(* CODESYS project templatecore.library
   Author: Multiple
   Placeholder: TemplateCore
   Title: TemplateCore
   Version: 2.0.0.2
   Description: Template Framework Code
   Company: TemplateCore Creators

Project tree, tasks and I/O mapping:
  libraries: Tc2_Standard, * (Beckhoff Automation GmbH); Tc2_System, * (Beckhoff Automation GmbH); Tc2_TcpIp, * (Beckhoff Automation GmbH); Tc2_Utilities, * (Beckhoff Automation GmbH); Tc3_Module, * (Beckhoff Automation GmbH)
  DUTs/
    Stats/
      data type Component_Stats
      data type StatsAggregateFIFOBuffer
      data type StatsAggregateRecord
      data type StatsConstants
      data type StatsEvent
      data type StatsEventFIFOBuffer
      data type StatsFailure
      data type StatsFailureFIFOBuffer
      data type StatsFault
      data type StatsFaultFIFOBuffer
      data type StatsShiftAggregateFIFOBuffer
      data type StatsShiftAggregateRecord
    data type Channels
    data type Colors
    data type ComponentIdentifier
    data type Dint100FIFOBuffer
    data type FaultMessage
    data type FrameWork
    data type FrameworkLocal
    data type GeneralMessage
    data type HMIBanner
    data type HMIMessage
    data type HMIMessageBuffer
    data type ID50FIFOBuffer
    data type LREAL100FIFOBuffer
    data type StateTimeStamp
    data type Station
    data type STRING256
    data type TimeStamp
    data type TraceFIFOBuffer
  GVLs/
    global variables GVL
  POUs/
    FrameWork/
      function F_AddMessage [ST]
      function F_FindMessage [ST]
      function block FB_Framework [ST]
      function block FIFO_HMIMessage [ST]: INIT, INSERT, PEEK, REMOVE
    OEE/
      function F_SendEvent [ST]
      function block FIFO_StatsAggregate [ST]: INIT, INSERT, PEEK, PEEKLAST, REMOVE
      function block FIFO_StatsEvent [ST]: INIT, INSERT, PEEK, REMOVE
      function block FIFO_StatsFailureLog [ST]: INIT, INSERT, PEEK, REMOVE
      function block FIFO_StatsFaultLog [ST]: INIT, INSERT, PEEK, REMOVE
      function block FIFO_StatsShiftAggregate [ST]: INIT, INSERT, PEEK, REMOVE
    StateTrace/
      function block FIFO_StateTrace [ST]: INIT, INSERT, PEEK, REMOVE
    TCP Communications/
      function block FB_TCPClient [ST]
    Utility/
      function F_GetTimeStamp [ST]
      function block FB_FileReadSettings [ST]
      function block FB_FileWriteSettings [ST]
      function block FB_Sensor [ST]
      function block FIFO_DINT100 [ST]: INIT, INSERT, PEEK, REMOVE
      function block FIFO_ID50 [ST]: INIT, INSERT, PEEK, REMOVE
      function block FIFO_LREAL100 [ST]: INIT, INSERT, PEEK, REMOVE
      function LEFTBigString [ST]
      function RIGHTBigString [ST]
    program MAIN [ST]
  Version/
    global variables Global_Version
  VISUs/
*)

// DUTs/Stats/Component_Stats
{attribute 'pack_mode' := '1'}
TYPE Component_Stats :
STRUCT
	AggregateInterval : DINT ; (*interval time in minutes*)
	PlannedDowntime : ARRAY [0..2] OF DINT;  (*index corresponds to shift number*)
	StartOfShift : ARRAY [0..2,0..1] OF DINT; (*[shift number],[hour,min]*)
	IdealCycleTime : LREAL; (*cycle time is second*)

	StatsEventFIFO : FIFO_StatsEvent := (Overwrite := TRUE);
	StatsEventBuffer : StatsEventFIFObuffer;
	StatsAggregateFIFO : FIFO_StatsAggregate := (Overwrite := TRUE);
	StatsAggregateBuffer : StatsAggregateFIFOBuffer;
	StatsShiftAggregateFIFO : FIFO_StatsShiftAggregate := (Overwrite := TRUE);
	StatsShiftAggregateBuffer : StatsShiftAggregateFIFOBuffer;
	StatsFaultLog : FIFO_StatsFaultLog := (Overwrite := TRUE);
	StatsFaultLogBuffer : StatsFaultFIFOBuffer;
	StatsFailureLog : FIFO_StatsFailureLog := (Overwrite := TRUE);
	StatsFailureLogBuffer : StatsFailureFIFOBuffer;

	StatsIdealCycleTimeFIFO : FIFO_LREAL100 := (Overwrite := FALSE);
	StatsIdealCycleTimeBuffer : LREAL100FIFOBuffer;
	StatsPartCountFIFO : FIFO_DINT100 := (Overwrite := FALSE);
	StatsPartCountBuffer : Dint100FIFOBuffer;

	Framework : Framework;
END_STRUCT
END_TYPE

// DUTs/Stats/StatsAggregateFIFOBuffer
TYPE StatsAggregateFIFOBuffer :
STRUCT
	Size:DINT := 864; (*3days at 5min*)
	Buffer:ARRAY [0..863] OF StatsAggregateRecord;
END_STRUCT
END_TYPE

// DUTs/Stats/StatsAggregateRecord
TYPE StatsAggregateRecord :
STRUCT
	TimeStamp : TimeStamp;
	OperatorStopTime : LREAL;
	OperatorStopCount : DINT;
	AutoStopTime:LREAL;
	AutoStopCount : DINT;
	WorkTime : LREAL;
	WorkCount: DINT;
	BypassTime: LREAL;
	BypassCount: DINT;
	BlockTime: LREAL;
	BlockCount: DINT;
	StarveTime:LREAL;
	StarveCount:DINT;
	FaultTime:LREAL;
	FaultCount:DINT;
	EmptyTime:LREAL;
	EmptyCount:DINT;
	RetryTime:LREAL;
	RetryCount:DINT;
	MasterTime:LREAL;
	MasterCount:DINT;
	OtherTime:LREAL;
	OtherCount:DINT;
	RejectCount:DINT;
	GoodCount:DINT;
	FirstTimeGoodCount:DINT;
	FirstTimeStartCount:DINT;
	GoodCycleTime:LREAL;
	InitCount:DINT;
	PartsForCurrentCycleTime: DINT;
	Shift : DINT;
END_STRUCT
END_TYPE

// DUTs/Stats/StatsConstants
TYPE StatsConstants :
STRUCT
	Aggregate :DINT := 1;

	OperatorStop : DINT := 100;
	MachineStop : DINT  :=101;
	Working : DINT := 102;
	Bypass : DINT := 103;
	Blocked : DINT := 104;
	Starved : DINT := 105;
	Faulted : DINT :=106;
	FaultAcknowledge : DINT := 107;
	Empty : DINT := 108;
	Retry : DINT := 109;
	Mastering : DINT := 110;

	Failure : DINT := 200;
	Good : DINT := 201;
	FirstTimeGood : DINT := 202;
	FirstTimeStart : DINT := 203;
	Initialize : DINT := 204;

	PartChange : DINT := 300;
	CycleTime : DINT := 301;


END_STRUCT
END_TYPE

// DUTs/Stats/StatsEvent
TYPE StatsEvent :
STRUCT
	TimeStamp : TimeStamp;
	EType : DINT;
	Data : ARRAY[0..4] OF REAL;
	StringData :ARRAY[0..3] OF STRING(80);
END_STRUCT
END_TYPE

// DUTs/Stats/StatsEventFIFOBuffer
{attribute 'pack_mode' := '1'}
TYPE StatsEventFIFOBuffer :
STRUCT
	Size:DINT := 100;
	Buffer:ARRAY[0..99] OF StatsEvent;
END_STRUCT
END_TYPE

// DUTs/Stats/StatsFailure
TYPE StatsFailure :
STRUCT
	TimeStamp : TimeStamp;
	StationID : DINT;
	FailureID : DINT;
	Parameters : STRING;
END_STRUCT
END_TYPE

// DUTs/Stats/StatsFailureFIFOBuffer
TYPE StatsFailureFIFOBuffer :
STRUCT
	Size:UDINT := 500;
	Buffer:ARRAY [0..499] OF StatsFailure;
END_STRUCT
END_TYPE

// DUTs/Stats/StatsFault
TYPE StatsFault:
STRUCT
	TimeStamp : TimeStamp;
	StationID : DINT;
	FaultID : DINT;
	AcknowledgeTime : LREAL;
	Duration : LREAL;
	Data : ARRAY [0..2] OF REAL;
	StringData : ARRAY [0..3] OF STRING;
END_STRUCT
END_TYPE

// DUTs/Stats/StatsFaultFIFOBuffer
TYPE StatsFaultFIFOBuffer :
STRUCT
	Size:UDINT := 500;
	Buffer:ARRAY [0..499] OF StatsFault;
END_STRUCT
END_TYPE

// DUTs/Stats/StatsShiftAggregateFIFOBuffer
TYPE StatsShiftAggregateFIFOBuffer :
STRUCT
	Size:DINT := 270; (*90 days*)
	Buffer:ARRAY [0..269] OF StatsShiftAggregateRecord;
END_STRUCT
END_TYPE

// DUTs/Stats/StatsShiftAggregateRecord
TYPE StatsShiftAggregateRecord :
STRUCT
	AggregateData : StatsAggregateRecord;
	Shift : DINT;
	ShiftStartTimeStamp : TimeStamp;
	AvailableTime : LREAL;
	NetAvailableTime : LREAL;
	TotalDownTime: LREAL;
	PlannedDownTime: LREAL;
	UnplannedDownTime: LREAL;
	OperatingTime : LREAL;
	EquipmentAvailability : LREAL;
	TotalParts: DINT;
	PerformanceEfficiency : LREAL;
	QualityRate : LREAL;
	OverallEquipmentEffectiveness :LREAL;
	CycleTimeAvgSum: LREAL;
	CycleTimeAvgCnt: DINT;
END_STRUCT
END_TYPE

// DUTs/Channels
TYPE Channels :
STRUCT
	Fault :DINT:= 1;
	Attention:DINT := 2;
	General:DINT:= 3;
	FirstFault:DINT:= 4;
END_STRUCT
END_TYPE

// DUTs/Colors
TYPE Colors :
STRUCT
	Red: DINT := 255;
	Green: DINT :=65280;
	Grey: DINT :=8421504;
	Black: DINT := 0;
	Yellow: DINT := 65535;
	Blue: DINT := 16711680;
	White:DINT := 16777215;
END_STRUCT
END_TYPE

// DUTs/ComponentIdentifier
TYPE ComponentIdentifier :
STRUCT
	ID:DINT;
	Name:STRING;
END_STRUCT
END_TYPE

// DUTs/Dint100FIFOBuffer
TYPE Dint100FIFOBuffer :
STRUCT
	Size:DINT := 100;
	Buffer:ARRAY [0..99] OF DINT;
END_STRUCT
END_TYPE

// DUTs/FaultMessage
TYPE FaultMessage :
STRUCT
	Id: DINT;
	Text: STRING256;
	AltText: STRING256;
END_STRUCT
END_TYPE

// DUTs/FrameWork
TYPE FrameWork :
STRUCT
	OnScan:BOOL;
	ResetStart:BOOL;
	ResetDone:BOOL;
	FullInitRequired:BOOL;
	Behavior:DINT;
	ComponentIDRecord: ComponentIdentifier;
END_STRUCT
END_TYPE

// DUTs/FrameworkLocal
TYPE FrameworkLocal :
STRUCT
	AsynchFault: BOOL;
	AsynchFaultReactionComplete: BOOL;
	Attention: BOOL;
	CycleAuto: BOOL;
	CycleFaulted: BOOL;
	CycleManual: BOOL;
	CycleReset: BOOL;
	ManualCycleRequested: BOOL;
	ManualCycleDone: BOOL;
	OKToStop: BOOL;
	SingleStepInhibit: BOOL;
	IgnorSingleStep: BOOL;
	FirstEntry: BOOL;
	LongFaultState: BOOL;
	CycleAutoFallingEdge: F_TRIG;
	CycleResetFallingEdge: F_TRIG;
	CycleManualFallingEdge: F_TRIG;
	State: DINT;
	NextState: DINT;
	LastAutoState: DINT;
	ReEntryState: DINT;
	FaultedState: DINT;
	FaultNumber: DINT;
	LocalFaultID: DINT;
	FullFaultID: DINT;
	tmrState: TON;
	tmrFault: TON;
	StateTimePreset:TIME;
	FaultTimePreset:TIME;
	FaultTimeLong: TIME;
	FaultTimeShort: TIME;
	FaultText: STRING256;
	FaultAltText: STRING256;
	FaultData:StatsFault;
	MsgText: STRING256;
	AltMsgText: STRING256;
	MsgArray: ARRAY [0..99] OF GeneralMessage;
	HMIMsg: HMIMessage;
	StateTimeStamp: StateTimeStamp;
	CurrentTime: TimeStamp;
	Name:STRING(30);
	AltName:STRING(30);
	pStateTraceBuffer: POINTER TO TraceFIFOBuffer;
	pStateTraceFifo: POINTER TO FIFO_StateTrace;
	pStats: POINTER TO Component_Stats;
END_STRUCT
END_TYPE

// DUTs/GeneralMessage
TYPE GeneralMessage :
STRUCT
	Id: DINT;
	BitNumber: DINT;
	Text: STRING;
	AltText:STRING;
END_STRUCT
END_TYPE

// DUTs/HMIBanner
TYPE HMIBanner :
STRUCT
	Text:STRING256;
	AltText:STRING256;
	Color:DINT;
END_STRUCT
END_TYPE

// DUTs/HMIMessage
TYPE HMIMessage :
STRUCT
	Channel: DINT;
	Color: DINT;
	Text: STRING256;
	AltText: STRING256;
END_STRUCT
END_TYPE

// DUTs/HMIMessageBuffer
TYPE HMIMessageBuffer :
STRUCT
	Size:DINT := 100;
	Buffer:ARRAY [0..99] OF HMIMessage;
END_STRUCT
END_TYPE

// DUTs/ID50FIFOBuffer
TYPE ID50FIFOBuffer :
STRUCT
	Size:DINT := 50;
	Buffer:ARRAY [0..49] OF ComponentIdentifier;
END_STRUCT
END_TYPE

// DUTs/LREAL100FIFOBuffer
TYPE LREAL100FIFOBuffer :
STRUCT
	Size:DINT := 100;
	Buffer:ARRAY [0..99] OF LREAL;
END_STRUCT
END_TYPE

// DUTs/StateTimeStamp
TYPE StateTimeStamp :
STRUCT
	Station:DINT;
	ID:DINT;
	State:DINT;
	TimeLo:UDINT;
	TimeHi:UDINT;
END_STRUCT
END_TYPE

// DUTs/Station
TYPE Station :
STRUCT
	CycleAuto:BOOL;
	CycleReset:BOOL;
	CycleManual:BOOL;
	CycleStopped:BOOL;
	CycleFaulted:BOOL;
	OKToStop:BOOL;
	OKForManual:BOOL;
	StopRequest:BOOL;
	EmergencyStop:BOOL;
	UnlatchFaults:BOOL;
	FaultReset:BOOL;
	FullInitRequired:BOOL;
	ResetDone:BOOL;
	SingleStep:BOOL;
	StepAdvance:BOOL;
	DryCycle:BOOL;
	Attention:BOOL;
	MachineStopRqst:BOOL;

	hiCycleStart:BOOL;
	hiCycleStop:BOOL;
	hiFaultAck:BOOL;
	hiFaultReset:BOOL;
	hiStationReset:BOOL;
	hiSingleStepOn:BOOL;
	hiSingleStepOff:BOOL;
	hiSingleStepAdvance:BOOL;
	hiManualMode:BOOL;
	hiLampTest:BOOL;
	hoStationResetRequired:BOOL;

	StationID:DINT;
	MachineID:DINT;
	FirstFault:StatsFault;
	PreviousStationID:DINT;
	NextStationID:DINT;
	HMIMessageFIFO: FIFO_HMIMessage;
	HMIMessageBuffer: HMIMessageBuffer;
	StationMessage:HMIBanner;
	OperatorMessage:HMIBanner;
	b500msPulse: BOOL;

	FaultedFIFO: FIFO_ID50;
	FaultedFIFOBuffer: ID50FIFOBuffer;
	NotOKtoStopFIFO: FIFO_ID50;
	NotOKToStopFIFOBuffer:ID50FIFOBuffer;
	AttentionRequiredFIFO: FIFO_ID50;
	AttentionRequiredFIFOBuffer: ID50FIFOBuffer;
	CycleManualFIFO: FIFO_ID50;
	CycleManualFIFOBuffer:ID50FIFOBuffer;

END_STRUCT
END_TYPE

// DUTs/STRING256
TYPE STRING256 :STRING[256];

END_TYPE

// DUTs/TimeStamp
TYPE TimeStamp :
STRUCT
	CurrentValue : T_ULarge_Integer;
	DateTime: TIMESTRUCT;
END_STRUCT
END_TYPE

// DUTs/TraceFIFOBuffer
TYPE TraceFIFOBuffer :
STRUCT
	Size:DINT := 1000;
	Buffer:ARRAY [0..999] OF StateTimeStamp;
END_STRUCT
END_TYPE

// GVLs/GVL
{attribute 'qualified_only'}
VAR_GLOBAL
	cColor:Colors;
	cChannel:Channels;
	cNullString:STRING;
	cEmptyHMIMessage: HMIMessage;(* ~(OPC:1:available for OPC-clients) *)
	gTimeZoneOffsetFromUTC: DINT := 0;
	gFirstScan:BOOL;
	gCurrentTime : TimeStamp;
END_VAR

// Version/Global_Version
{attribute 'TcGenerated'}
// This function has been automatically generated from the project information.
VAR_GLOBAL CONSTANT
	{attribute 'const_non_replaced'}
	{attribute 'linkalways'}
	stLibVersion_TemplateCore : ST_LibVersion := (iMajor := 2, iMinor := 0, iBuild := 0, iRevision := 2, sVersion := '2.0.0.2');
END_VAR

// POUs/FrameWork/F_AddMessage
FUNCTION F_AddMessage : BOOL
VAR_INPUT
	pStation:  POINTER TO Station;
	Text:STRING256	;
	AltText:STRING256;
	Color:DINT;
	Channel:DINT;
END_VAR
VAR
	StationAddress:DINT;
	HMIMsg:HMIMessage;

END_VAR

HMIMsg.Text := Text;
HMIMsg.AltText := AltText;
HMIMsg.Color := Color;
HMIMsg.Channel := Channel;
pStation^.HMIMessageFIFO.INSERT(pFIFO:=ADR(pStation^.HMIMessageBuffer), in :=HMIMsg);

END_FUNCTION

// POUs/FrameWork/F_FindMessage
FUNCTION F_FindMessage : GeneralMessage
VAR_INPUT
	pLocal: POINTER TO FrameworkLocal;
	State:DINT;
	ID: DINT;
END_VAR
VAR
	Msg:GeneralMessage;
	idx:DINT;
	length:DINT;
END_VAR

length := SIZEOF(pLocal^.MsgArray) / SIZEOF(Msg);
Msg.Text  :='**No message text**';
Msg.AltText :='**No alt message text**';
FOR idx :=0 TO (length-1) DO
	IF pLocal^.MsgArray[idx].Id = (State * 10 + ID) THEN
		Msg := pLocal^.MsgArray[idx];
		EXIT;
	END_IF
END_FOR
F_FindMessage := Msg;

END_FUNCTION

// POUs/FrameWork/FB_Framework
FUNCTION_BLOCK FB_Framework
VAR_INPUT
	pFrameWork: POINTER TO FrameWork;
	pLocal: POINTER TO FrameworkLocal;
	pStation: POINTER TO Station;
END_VAR

VAR_OUTPUT
END_VAR

VAR
	InitialScan: R_TRIG;
	ActiveStationID: DINT;
	Msg:GeneralMessage;
	cChannel: Channels;
END_VAR

VAR_STAT CONSTANT
	cColor: Colors;
END_VAR

(****************************************************************************
* Framework Post-Sequence Logic, DO NOT modify this section *
*****************************************************************************)

InitialScan(CLK := TRUE);
IF InitialScan.Q THEN
        pLocal^.State := 9999;
        pLocal^.NextState := 5000;
END_IF

(*  Fault Logic  *)
pLocal^.tmrFault(IN := (NOT pLocal^.OKToStop AND NOT pLocal^.FirstEntry AND NOT pLocal^.SingleStepInhibit  AND
				(pLocal^.CycleAuto OR pLocal^.CycleReset OR pLocal^.CycleManual)), PT := pLocal^.FaultTimePreset);
IF pLocal^.FaultNumber  > 0 THEN
	IF  NOT pLocal^.CycleFaulted THEN
		pLocal^.CycleFaulted := TRUE;
		pLocal^.FaultedState := pLocal^.state;
		IF (NOT pLocal^.AsynchFault) OR pLocal^.AsynchFaultReactionComplete THEN
			Msg := F_FindMessage(pLocal,  pLocal^.State, pLocal^.FaultNumber);
			pLocal^.FaultData.FaultID := pFrameWork^.ComponentIDRecord.ID * 100000 + pLocal^.state*10 + pLocal^.FaultNumber;
		ELSE
			Msg := F_FindMessage(pLocal,  0, pLocal^.FaultNumber);
			pLocal^.FaultData.FaultID := pFrameWork^.ComponentIDRecord.ID * 100000 + pLocal^.FaultNumber;
		END_IF
		pLocal^.MsgText :=  'Fault: ';
		pLocal^.AltMsgText  := 'AltFault: ';
		pLocal^.MsgText := CONCAT(pLocal^.MsgText,DINT_TO_STRING(pLocal^.FaultData.FaultID));
		pLocal^.MsgText := CONCAT(pLocal^.MsgText,' ');
		pLocal^.MsgText := CONCAT(pLocal^.MsgText, pLocal^.Name);
		pLocal^.MsgText := CONCAT(pLocal^.MsgText,' -  ');
		pLocal^.MsgText := CONCAT(pLocal^.MsgText, Msg.Text);
		pLocal^.AltMsgText := CONCAT(pLocal^.AltMsgText,DINT_TO_STRING(pLocal^.FaultData.FaultID));
		pLocal^.AltMsgText := CONCAT(pLocal^.AltMsgText,' ');
		pLocal^.AltMsgText := CONCAT(pLocal^.AltMsgText, pLocal^.AltName);
		pLocal^.AltMsgText := CONCAT(pLocal^.MsgText,' -  ');
		pLocal^.AltMsgText:=CONCAT(pLocal^.AltMsgText, Msg.AltText);
		F_AddMessage(pStation, pLocal^.MsgText, pLocal^.AltMsgText, cColor.Red, cChannel.Fault);
		IF pStation^.FirstFault.FaultID = 0 THEN
			pStation^.FirstFault := pLocal^.FaultData;
			pStation^.FirstFault.StationID  := pStation^.StationID;
			pStation^.FirstFault.StringData[0] :=pLocal^.MsgText;
			pStation^.FirstFault.StringData[1] :=pLocal^.AltMsgText;
		END_IF
	END_IF
END_IF

(*END fault logic*)

(***************************************************************************
* Framework Pre-Sequence Logic, DO NOT modify this section *
****************************************************************************)

IF pLocal^.NextState <> pLocal^.state THEN
	pLocal^.FirstEntry := TRUE;
	pLocal^.state := pLocal^.NextState;
	pLocal^.tmrState(IN:=FALSE); (*clear timer if state changes*)

	pLocal^.CurrentTime := GVL.gCurrentTime;
	pLocal^.StateTimeStamp.ID := pFrameWork^.ComponentIDRecord.ID;
	pLocal^.StateTimeStamp.State := pLocal^.State;
	pLocal^.StateTimeStamp.TimeHi := pLocal^.CurrentTime.CurrentValue.dwHighPart;
	pLocal^.StateTimeStamp.TimeLo:= pLocal^.CurrentTime.CurrentValue.dwLowPart;
	pLocal^.pStateTraceFifo^.INSERT(pFIFO := pLocal^.pStateTraceBuffer, in := pLocal^.StateTimeStamp);
ELSE
	pLocal^.FirstEntry := FALSE;
	pLocal^.tmrState(IN:=TRUE,PT:=pLocal^.StateTimePreset);
END_IF

(*On the falling edge of CycleAuto, grab the current state as LastAutoState.
    Also, set the default ReEntryState to the LastAutoState so that we pick back up where 
    we left off after a simple cycle stop / cycle start.
    Set State to 5000, the Idle state. *)

pLocal^.CycleAutoFallingEdge(CLK:=pLocal^.CycleAuto);
IF pLocal^.CycleAutoFallingEdge.Q THEN
	pLocal^.LastAutoState := pLocal^.State;
	pLocal^.ReEntryState := pLocal^.LastAutoState;
	pLocal^.NextState := 5000;
END_IF

(* On the falling edge of CycleReset, set State to 5000, the Idle state.   *)
pLocal^.CycleResetFallingEdge(Clk:=pLocal^.CycleReset);
IF pLocal^.CycleResetFallingEdge.Q THEN
	pLocal^.NextState := 5000;
END_IF

(* On the falling edge of CycleManual, set State to 5000, the Idle state.  *)
pLocal^.CycleManualFallingEdge(Clk:=pLocal^.CycleManual);
IF pLocal^.CycleManualFallingEdge.Q THEN
	pLocal^.NextState := 5000;
END_IF

pLocal^.CycleAuto:=pStation^.CycleAuto AND NOT pLocal^.CycleFaulted;
pLocal^.CycleReset := pStation^.CycleReset AND NOT pLocal^.CycleFaulted;
pLocal^.CycleManual := pLocal^.ManualCycleRequested AND (NOT pLocal^.ManualCycleDone) AND (NOT pStation^.CycleFaulted);
pLocal^.SingleStepInhibit := pStation^.SingleStep AND NOT pStation^.StepAdvance AND NOT pLocal^.IgnorSingleStep;

IF pStation^.UnlatchFaults THEN
	pLocal^.CycleFaulted := FALSE;
	pLocal^.FaultNumber := 0;
END_IF

IF pLocal^.CycleFaulted THEN
	pStation^.FaultedFIFO.INSERT(pFIFO := ADR(pStation^.FaultedFIFOBuffer), in:=pFrameWork^.ComponentIDRecord);
END_IF
IF pLocal^.CycleManual THEN
	pStation^.CycleManualFIFO.INSERT(pFIFO := ADR(pStation^.CycleManualFIFOBuffer), in:=pFrameWork^.ComponentIDRecord);
END_IF
IF pLocal^.Attention THEN
	pStation^.AttentionRequiredFIFO.INSERT(pFIFO := ADR(pStation^.AttentionRequiredFIFOBuffer), in:=pFrameWork^.ComponentIDRecord);
END_IF
IF NOT pLocal^.OKToStop THEN
	pStation^.NotOKtoStopFIFO.INSERT(pFIFO := ADR(pStation^.NotOKtoStopFIFOBuffer), in:=pFrameWork^.ComponentIDRecord);
END_IF
pLocal^.OKToStop := FALSE;
(*END of framework*)

END_FUNCTION_BLOCK

// POUs/FrameWork/FIFO_HMIMessage
FUNCTION_BLOCK FIFO_HMIMessage
VAR_INPUT
	Overwrite	: BOOL;
	pFIFO		: POINTER TO HMIMessageBuffer;
	in			: HMIMessage;
END_VAR
VAR_OUTPUT
	Err		: BOOL;
	Count	: DINT;
	Full		: BOOL;
	out		: HMIMessage;
END_VAR
VAR
	Head : DINT;
	Tail: DINT;
	Idx: DINT;
END_VAR

;

ACTION INIT:
idx := pFIFO^.Size * SIZEOF(in);
MEMSET(ADR( pFIFO^.Buffer[0]), 0, DINT_TO_UDINT(idx));
MEMSET(ADR(in),0,SIZEOF(in));
MEMSET(ADR(out),0,SIZEOF(out));
Count:=0;
Head:=0;
Tail:=0;
Full:=0;
Err:=0;
END_ACTION

ACTION INSERT:
Err := 0;
IF (Full AND Overwrite) OR NOT Full THEN
	pFIFO^.buffer[Head]:=in;
	Head := Head + 1;
	IF Head = pFIFO^.Size THEN
		Head:=0;
	END_IF
	IF Full THEN
		Tail := Tail +1;
		IF Tail = pFIFO^.Size THEN
			Tail :=0;
		END_IF
	ELSE
		Count := Count  +1;
	END_IF
ELSE
	err:=1;
END_IF
Full := (Head = Tail);
END_ACTION

ACTION PEEK:
err:=0;
IF Full OR (Tail <> Head) THEN
	out := pFIFO^.buffer[Tail];
ELSE
	err:=1; (*fifo is empty*)
END_IF
END_ACTION

ACTION REMOVE:
err:=0;
IF NOT Full AND (Head = Tail) THEN
	(*empty*)
	err:=1;
ELSE
	out := pFIFO^.Buffer[Tail];
	MEMSET(ADR(pFIFO^.buffer[Tail]), 0, SIZEOF (in));
	Tail := Tail +1;
	Count := Count  - 1;
	IF Tail = pFIFO^.Size THEN
		Tail := 0;
	END_IF
	Full := 0;
END_IF
END_ACTION

END_FUNCTION_BLOCK

// POUs/OEE/F_SendEvent
FUNCTION F_SendEvent : BOOL
VAR_INPUT
	pStatsFIFO	: POINTER TO FIFO_StatsEvent;
	pBuffer		: POINTER TO StatsEventFIFOBuffer;
	pEvent		: POINTER TO StatsEvent;
END_VAR
VAR
	CurrentTime: TimeStamp;
END_VAR

pEvent^.TimeStamp:= GVL.gCurrentTime;
pStatsFIFO^.INSERT(pFIFO:=pBuffer, in:= pEvent^);
MEMSET(pEvent,0,SIZEOF(pEvent^));

END_FUNCTION

// POUs/OEE/FIFO_StatsEvent
{attribute 'pack_mode' := '1'}
FUNCTION_BLOCK FIFO_StatsEvent
VAR_INPUT
	Overwrite	: BOOL;
	pFIFO		: POINTER TO StatsEventFIFOBuffer;
	in			: StatsEvent;
END_VAR
VAR_OUTPUT
	Err		: BOOL;
	Count	: DINT;
	Full		: BOOL;
	out		: StatsEvent;
END_VAR
VAR
	Head : DINT;
	Tail: DINT;
	Idx: DINT;
END_VAR

ACTION INIT:
Idx := pFIFO^.Size * SIZEOF(in);
MEMSET(ADR( pFIFO^.Buffer[0]), 0, DINT_TO_UDINT(idx));
MEMSET(ADR(in),0,SIZEOF(in));
MEMSET(ADR(out),0,SIZEOF(out));
Count:=0;
Head:=0;
Tail:=0;
Full:=0;
Err:=0;
END_ACTION

ACTION INSERT:
Err := 0;
IF (Full AND Overwrite) OR NOT Full THEN
	pFIFO^.buffer[Head]:=in;
	Head := Head + 1;
	IF Head = pFIFO^.Size THEN
		Head:=0;
	END_IF
	IF Full THEN
		Tail := Tail +1;
		IF Tail = pFIFO^.Size THEN
			Tail :=0;
		END_IF
	ELSE
		Count := Count  +1;
	END_IF
ELSE
	err:=1;
END_IF
Full := (Head = Tail);
END_ACTION

ACTION PEEK:
err:=0;
IF Full OR (Tail <> Head) THEN
	out := pFIFO^.buffer[Tail];
ELSE
	err:=1; (*fifo is empty*)
END_IF
END_ACTION

ACTION REMOVE:
err:=0;
IF NOT Full AND (Head = Tail) THEN
	(*empty*)
	err:=1;
ELSE
	out := pFIFO^.Buffer[Tail];
	MEMSET(ADR(pFIFO^.buffer[Tail]), 0, SIZEOF (in));
	Tail := Tail +1;
	Count := Count  - 1;
	IF Tail = pFIFO^.Size THEN
		Tail := 0;
	END_IF
	Full := 0;
END_IF
END_ACTION

END_FUNCTION_BLOCK

// POUs/OEE/FIFO_StatsAggregate
{attribute 'pack_mode' := '1'}
FUNCTION_BLOCK FIFO_StatsAggregate
VAR_INPUT
	Overwrite	: BOOL;
	pFIFO		: POINTER TO StatsAggregateFIFOBuffer;
	in			: StatsAggregateRecord;
END_VAR
VAR_OUTPUT
	Err		: BOOL;
	Count	: DINT;
	Full		: BOOL;
	out		: StatsAggregateRecord;
END_VAR
VAR
	Head : DINT;
	Tail: DINT;
	Idx: DINT;
END_VAR

ACTION INIT:
idx := pFIFO^.Size * SIZEOF(in);
MEMSET(ADR( pFIFO^.Buffer[0]), 0, DINT_TO_UDINT(idx));
MEMSET(ADR(in),0,SIZEOF(in));
MEMSET(ADR(out),0,SIZEOF(out));
Count:=0;
Head:=0;
Tail:=0;
Full:=0;
Err:=0;
END_ACTION

ACTION INSERT:
Err := 0;
IF (Full AND Overwrite) OR NOT Full THEN
	pFIFO^.buffer[Head]:=in;
	Head := Head + 1;
	IF Head = pFIFO^.Size THEN
		Head:=0;
	END_IF
	IF Full THEN
		Tail := Tail +1;
		IF Tail = pFIFO^.Size THEN
			Tail :=0;
		END_IF
	ELSE
		Count := Count  +1;
	END_IF
ELSE
	err:=1;
END_IF
Full := (Head = Tail);
END_ACTION

ACTION PEEK:
err:=0;
IF Full OR (Tail <> Head) THEN
	out := pFIFO^.buffer[Head];
ELSE
	err:=1; (*fifo is empty*)
END_IF
END_ACTION

ACTION PEEKLAST:
err:=0;
IF Full OR (Tail <> Head) THEN
	out := pFIFO^.buffer[Tail];
ELSE
	err:=1; (*fifo is empty*)
END_IF
END_ACTION

ACTION REMOVE:
err:=0;
IF NOT Full AND (Head = Tail) THEN
	(*empty*)
	err:=1;
ELSE
	out := pFIFO^.Buffer[Tail];
	MEMSET(ADR(pFIFO^.buffer[Tail]), 0, SIZEOF (in));
	Tail := Tail +1;
	Count := Count  - 1;
	IF Tail = pFIFO^.Size THEN
		Tail := 0;
	END_IF
	Full := 0;
END_IF
END_ACTION

END_FUNCTION_BLOCK

// POUs/OEE/FIFO_StatsFailureLog
FUNCTION_BLOCK FIFO_StatsFailureLog
VAR_INPUT
	Overwrite	: BOOL;
	pFIFO		: POINTER TO StatsFailureFIFOBuffer;
	in			: StatsFailure;
END_VAR
VAR_OUTPUT
	Err		: BOOL;
	Count	: DINT;
	Full		: BOOL;
	out		: StatsFailure;
END_VAR
VAR
	Head : DINT;
	Tail: DINT;
	Idx: DINT;
END_VAR

ACTION INIT:
idx := UDINT_TO_DINT(pFIFO^.Size * SIZEOF(in));
MEMSET(ADR( pFIFO^.Buffer[0]), 0, DINT_TO_UDINT(idx));
MEMSET(ADR(in),0,SIZEOF(in));
MEMSET(ADR(out),0,SIZEOF(out));
Count:=0;
Head:=0;
Tail:=0;
Full:=0;
Err:=0;
END_ACTION

ACTION INSERT:
Err := 0;
IF (Full AND Overwrite) OR NOT Full THEN
	pFIFO^.buffer[Head]:=in;
	Head := Head + 1;
	IF Head = UDINT_TO_DINT(pFIFO^.Size) THEN
		Head:=0;
	END_IF
	IF Full THEN
		Tail := Tail +1;
		IF Tail = UDINT_TO_DINT(pFIFO^.Size) THEN
			Tail :=0;
		END_IF
	ELSE
		Count := Count  +1;
	END_IF
ELSE
	err:=1;
END_IF
Full := (Head = Tail);
END_ACTION

ACTION PEEK:
err:=0;
IF Full OR (Tail <> Head) THEN
	out := pFIFO^.buffer[Tail];
ELSE
	err:=1; (*fifo is empty*)
END_IF
END_ACTION

ACTION REMOVE:
err:=0;
IF NOT Full AND (Head = Tail) THEN
	(*empty*)
	err:=1;
ELSE
	out := pFIFO^.Buffer[Tail];
	MEMSET(ADR(pFIFO^.buffer[Tail]), 0, SIZEOF (in));
	Tail := Tail +1;
	Count := Count  - 1;
	IF Tail = UDINT_TO_DINT(pFIFO^.Size) THEN
		Tail := 0;
	END_IF
	Full := 0;
END_IF
END_ACTION

END_FUNCTION_BLOCK

// POUs/OEE/FIFO_StatsFaultLog
FUNCTION_BLOCK FIFO_StatsFaultLog
VAR_INPUT
	Overwrite	: BOOL;
	pFIFO		: POINTER TO StatsFaultFIFOBuffer;
	in			: StatsFault;
END_VAR
VAR_OUTPUT
	Err		: BOOL;
	Count	: DINT;
	Full		: BOOL;
	out		: StatsFault;
END_VAR
VAR
	Head : DINT;
	Tail: DINT;
	Idx: DINT;
END_VAR

ACTION INIT:
idx := UDINT_TO_DINT(pFIFO^.Size * SIZEOF(in));
MEMSET(ADR( pFIFO^.Buffer[0]), 0, DINT_TO_UDINT(idx));
MEMSET(ADR(in),0,SIZEOF(in));
MEMSET(ADR(out),0,SIZEOF(out));
Count:=0;
Head:=0;
Tail:=0;
Full:=0;
Err:=0;
END_ACTION

ACTION INSERT:
Err := 0;
IF (Full AND Overwrite) OR NOT Full THEN
	pFIFO^.buffer[Head]:=in;
	Head := Head + 1;
	IF Head = UDINT_TO_DINT(pFIFO^.Size) THEN
		Head:=0;
	END_IF
	IF Full THEN
		Tail := Tail +1;
		IF Tail = UDINT_TO_DINT(pFIFO^.Size) THEN
			Tail :=0;
		END_IF
	ELSE
		Count := Count  +1;
	END_IF
ELSE
	err:=1;
END_IF
Full := (Head = Tail);
END_ACTION

ACTION PEEK:
err:=0;
IF Full OR (Tail <> Head) THEN
	out := pFIFO^.buffer[Tail];
ELSE
	err:=1; (*fifo is empty*)
END_IF
END_ACTION

ACTION REMOVE:
err:=0;
IF NOT Full AND (Head = Tail) THEN
	(*empty*)
	err:=1;
ELSE
	out := pFIFO^.Buffer[Tail];
	MEMSET(ADR(pFIFO^.buffer[Tail]), 0, SIZEOF (in));
	Tail := Tail +1;
	Count := Count  - 1;
	IF Tail = UDINT_TO_DINT(pFIFO^.Size) THEN
		Tail := 0;
	END_IF
	Full := 0;
END_IF
END_ACTION

END_FUNCTION_BLOCK

// POUs/OEE/FIFO_StatsShiftAggregate
FUNCTION_BLOCK FIFO_StatsShiftAggregate
VAR_INPUT
	Overwrite	: BOOL;
	pFIFO		: POINTER TO StatsShiftAggregateFIFOBuffer;
	in			: StatsShiftAggregateRecord;
	PeekCnt		: DINT;
END_VAR
VAR_OUTPUT
	Err		: BOOL;
	Count	: DINT;
	Full		: BOOL;
	out		: StatsShiftAggregateRecord;
END_VAR
VAR
	Head : DINT;
	Tail: DINT;
	Idx: DINT;

	PeekHead: DINT;
	PeekTail: DINT;
END_VAR

ACTION INIT:
idx := pFIFO^.Size * SIZEOF(in);
MEMSET(ADR( pFIFO^.Buffer[0]), 0, DINT_TO_UDINT(idx));
MEMSET(ADR(in),0,SIZEOF(in));
MEMSET(ADR(out),0,SIZEOF(out));
Count:=0;
Head:=0;
Tail:=0;
Full:=0;
Err:=0;
END_ACTION

ACTION INSERT:
idx := (pFIFO^.Size) * SIZEOF(in);
MEMSET(ADR( pFIFO^.Buffer[0]), 0, DINT_TO_UDINT(idx));
MEMSET(ADR(in),0,SIZEOF(in));
MEMSET(ADR(out),0,SIZEOF(out));
Count:=0;
Head:=0;
Tail:=0;
Full:=0;
Err:=0;
END_ACTION

ACTION PEEK:
err:=0;

PeekHead := Head;
PeekTail := Tail;
FOR Idx := 0 TO PeekCnt DO

	IF NOT Full AND (PeekHead = PeekTail) THEN
		(*empty*)
		err:=1;
	ELSE
		out := pFIFO^.Buffer[PeekTail];
		PeekTail := PeekTail +1;

		IF PeekTail = pFIFO^.Size THEN
			PeekTail := 0;
		END_IF
		Full := 0;
	END_IF
END_FOR

PeekCnt := 0;
END_ACTION

ACTION REMOVE:
err:=0;
IF NOT Full AND (Head = Tail) THEN
	(*empty*)
	err:=1;
ELSE
	out := pFIFO^.Buffer[Tail];
	MEMSET(ADR(pFIFO^.buffer[Tail]), 0, SIZEOF (in));
	Tail := Tail +1;
	Count := Count  - 1;
	IF Tail = pFIFO^.Size THEN
		Tail := 0;
	END_IF
	Full := 0;
END_IF
END_ACTION

END_FUNCTION_BLOCK

// POUs/StateTrace/FIFO_StateTrace
FUNCTION_BLOCK FIFO_StateTrace
VAR_INPUT
	Overwrite	: BOOL;
	pFIFO		: POINTER TO TraceFIFOBuffer;
	in			: StateTimeStamp;
END_VAR
VAR_OUTPUT
	Err		: BOOL;
	Count	: DINT;
	Full		: BOOL;
	out		: StateTimeStamp;
END_VAR
VAR
	Head : DINT;
	Tail: DINT;
	Idx: DINT;
END_VAR

ACTION INIT:
idx := pFIFO^.Size * SIZEOF(in);
MEMSET(ADR( pFIFO^.Buffer[0]), 0, DINT_TO_UDINT(idx));
MEMSET(ADR(in),0,SIZEOF(in));
MEMSET(ADR(out),0,SIZEOF(out));
Count:=0;
Head:=0;
Tail:=0;
Full:=0;
Err:=0;
END_ACTION

ACTION INSERT:
Err := 0;
IF (Full AND Overwrite) OR NOT Full THEN
	pFIFO^.buffer[Head]:=in;
	Head := Head + 1;
	IF Head = pFIFO^.Size THEN
		Head:=0;
	END_IF
	IF Full THEN
		Tail := Tail +1;
		IF Tail = pFIFO^.Size THEN
			Tail :=0;
		END_IF
	ELSE
		Count := Count  +1;
	END_IF
ELSE
	err:=1;
END_IF
Full := (Head = Tail);
END_ACTION

ACTION PEEK:
err:=0;
IF Full OR (Tail <> Head) THEN
	out := pFIFO^.buffer[Tail];
ELSE
	err:=1; (*fifo is empty*)
END_IF
END_ACTION

ACTION REMOVE:
err:=0;
IF NOT Full AND (Head = Tail) THEN
	(*empty*)
	err:=1;
ELSE
	out := pFIFO^.Buffer[Tail];
	MEMSET(ADR(pFIFO^.buffer[Tail]), 0, SIZEOF (in));
	Tail := Tail +1;
	Count := Count  - 1;
	IF Tail = pFIFO^.Size THEN
		Tail := 0;
	END_IF
	Full := 0;
END_IF
END_ACTION

END_FUNCTION_BLOCK

// POUs/TCP Communications/FB_TCPClient
FUNCTION_BLOCK FB_TCPClient
VAR_INPUT
	sRemoteHost: STRING(15);
	nRemotePort:UDINT;
	bConnect:BOOL;
	bSend:BOOL;
	bReceived:BOOL;
	bClearError: BOOL;
	bFlush : BOOL;
	pReceiveBuffer : POINTER TO ARRAY[0..4095] OF USINT;
	pTransmitBuffer : POINTER TO ARRAY[0..4095] OF USINT;
	TransmitLength : DINT;
	pMessageEOF : POINTER TO ARRAY [0..11] OF USINT;
	EOFLength : DINT;
	MessageLength : DINT;
END_VAR
VAR_OUTPUT
	bConnected:BOOL;
	bTransmitComplete:BOOL;
	bError:BOOL;
	bDataAvailable:BOOL;
	nErrorID:DINT;
	sErrorText:STRING(80);
	nReceiveLength:DINT;
	bFlushComplete : BOOL;
END_VAR
VAR
	(*Standard Framework Tags*)
	State: DINT;
	LastState: DINT;
	FaultNumber: DINT;
	FaultedState: DINT;
	FirstEntry: BOOL;
	tmrState: TON;
	MsgText: STRING256;
	AltMsgText:STRING256;
	(*End of Standard Framework Tags*)

	MsgIn: ARRAY[0..4095] OF USINT; (*STRING(4096);*)
	InBuffer: ARRAY[0..12287] OF USINT; (*STRING(12288);*)
	TempBuffer:ARRAY[0..12287] OF USINT;
	InBufferDataLength:DINT :=0;
	pInBuffer:POINTER TO STRING(12288); (*used only to view data easier for debug*)
  	tState120Timer:TON;
	tState200Timer:TON;
	tState500Timer:TON;
	Mode : DINT;
	index : DINT;
	EOFIndex : DINT;
	FindState : DINT;

	hSocketHandle:T_HSOCKET;
	fbSocketConnect : FB_SocketConnect;
	fbSocketClose : FB_SocketClose;
	fbSocketCloseAll : FB_SocketCloseAll;
	fbSocketReceive :FB_SocketReceive;
	fbSocketSend :FB_SocketSend;

END_VAR

VAR CONSTANT
	cEOF : DINT := 1;
	cFixedLength :DINT := 2;
	cContinuous : DINT := 3;
END_VAR

(*If State Change, capture rising edge with FirstEntry.*)
IF State <> LastState THEN
	FirstEntry := TRUE;
	tmrState(IN:=FALSE); (*clear timer if state changes*)
	LastState := State;
ELSIF FirstEntry THEN
	FirstEntry := FALSE;
END_IF

IF EOFLength > 0 THEN
	Mode := cEOF;
ELSIF MessageLength > 0 THEN
	Mode := cFixedLength;
ELSE
	Mode := cContinuous;
END_IF


(**********************
* Sequence logic  *
***********************)
CASE State OF

0:	(*Idle*)
	IF FirstEntry THEN
		bConnected := FALSE;
		bDataAvailable := FALSE;
		bFlushComplete := FALSE;
	END_IF
	IF bConnect AND NOT bError THEN
		State := 100;
	ELSIF bClearError THEN
		bError := FALSE;
		nErrorID := 0;
		sErrorText := GVL.cNullString;
	END_IF

100:	(*Check Parameters*)
	IF sRemoteHost = GVL.cNullString OR nRemotePort = 0 THEN
		bError := TRUE;
		sErrorText:='Invalid connect parameters';
	END_IF
	IF NOT bError THEN
		State := 110;
	ELSE
		State := 0;
	END_IF

110:	(*Connect*)
	IF FirstEntry THEN
		fbSocketConnect(bExecute := FALSE);
		fbSocketConnect(
			sSrvNetId := GVL.cNullString,
			sRemoteHost := sRemoteHost,
			nRemotePort := nRemotePort,
			bExecute := TRUE,
			tTimeout := T#15s  );
	END_IF
	IF fbSocketConnect.bBusy THEN
		State := 120;
	END_IF

120:	(*Wait For Connection*)
	tmrState(IN:=TRUE , PT:=T#4s );
	fbSocketConnect(bExecute:= FALSE);
	IF NOT fbSocketConnect.bBusy  THEN
		IF  fbSocketConnect.bError THEN
			bError := TRUE;
			sErrorText:= 'Socket Connection Could Not Be Made To ';
			sErrorText := CONCAT(sErrorText, sRemoteHost);
			sErrorText := CONCAT(sErrorText,  ' Port ');
 			sErrorText := CONCAT(sErrorText,  UDINT_TO_STRING(nRemotePort));
			State := 500;
		ELSE
			IF fbSocketConnect.hSocket.handle > 0 THEN
				hSocketHandle := fbSocketConnect.hSocket;
				bConnected := TRUE;
				State := 600; (*clear all buffer first*)
			END_IF
		END_IF
	ELSE
		IF tmrState.Q THEN
			bError := TRUE;
			sErrorText := 'Socket Connection Timed Out: ';
			sErrorText := CONCAT(sErrorText, sRemoteHost);
			sErrorText := CONCAT(sErrorText,  ' Port ');
 			sErrorText := CONCAT(sErrorText,  UDINT_TO_STRING(nRemotePort));
			State := 500;
		END_IF
	END_IF

200: (*Connected*)
	IF NOT bConnect THEN
		State := 500;
	END_IF
	IF bReceived  THEN
		State := 300;
	END_IF
	IF bSend THEN
		State := 400;
	END_IF
	IF bFlush THEN
		State := 600;
	END_IF

	tmrState(IN:=TRUE,PT:=t#100ms);
	IF tmrState.Q AND State = 200 THEN
		(*Poll for incomming packet*)
		State := 210;
		(* ejm - moved this from state 210 because it needs one PLC Scan *)
		fbSocketReceive(bExecute:=FALSE);
	END_IF

210:	(*Receive Data If Any*)
	IF FirstEntry THEN
		fbSocketReceive(
			sSrvNetId := GVL.cNullString,
			hSocket := hSocketHandle ,
			cbLen := SIZEOF(MsgIn),
			pDest := ADR(MsgIn),
			bExecute := TRUE,
			tTimeout := T#5s );
	END_IF
	IF NOT FirstEntry AND fbSocketReceive.bBusy THEN
		State := 220;
	END_IF

220:	(*Wait For Return*)
	fbSocketReceive(bExecute:=FALSE);
	IF NOT  fbSocketReceive.bBusy THEN
		IF NOT fbSocketReceive.bError THEN
			IF fbSocketReceive.nRecBytes > 0 THEN
				State := 230;
			ELSE
				State := 200;
			END_IF
		ELSE
			bError := 1;
			sErrorText := 'Socket Receive Error: ';
			sErrorText := CONCAT(sErrorText, sRemoteHost);
			sErrorText := CONCAT(sErrorText,  ' Port ');
 			sErrorText := CONCAT(sErrorText,  UDINT_TO_STRING(nRemotePort));
			State := 500;
		END_IF
	END_IF

230: (*copy packet data*)

	IF (UDINT_TO_DINT(fbSocketReceive.nRecBytes) + InBufferDataLength) <= SIZEOF(Inbuffer) THEN
		(*data will fit in buffer*)
		MEMCPY(ADR(InBuffer[InBufferDataLength]),ADR(MsgIn),fbSocketReceive.nRecBytes);
		InBufferDataLength := InBufferDataLength +UDINT_TO_DINT(fbSocketReceive.nRecBytes);
		MEMSET(ADR(MsgIn),0,SIZEOF(MsgIn)); (* Clear MsgIn so longer messages don't remain after fbSocketReceive*)
		State := 240;
	ELSE
		bError:=1;
		sErrorText:='Buffer Overflow';
		State := 500;
	END_IF

240: (*Search Message*)

	CASE Mode OF

		cEOF:	(*search for eof*)

			pInBuffer := ADR(InBuffer[0]); (*just for reference. Makes looking at data easier*)
			IF NOT bDataAvailable THEN
				(*search buffer for EOF string*)
				FindState:=0; (*index for counting successive matches to EOF*)
				FOR index :=0 TO InBufferDataLength - 1 DO
					IF InBuffer[index] = pMessageEOF^[FindState] THEN
						(*match found*)
						FindState := FindState + 1;
						IF findState = EOFLength THEN
							EOFIndex:=index - EOFLength +1;
							EXIT;
						END_IF
					ELSE
						IF FindState > 0 THEN
							FindState:=0; (*reset counter and start looking for new match*)
							IF InBuffer[index] = pMessageEOF^[FindState] THEN (*must check current index for match to first element of EOF.*)
								FindState:=1;
							END_IF
						END_IF
					END_IF
				END_FOR;
			END_IF
			IF EOFIndex >0 THEN (*message found*)
				MEMCPY(pReceiveBuffer, ADR(InBuffer[0]),DINT_TO_UDINT((EOFIndex + EOFLength))); (*copy message up to AND including EOF into receive message*)
				Index := EOFIndex + EOFLength;
				nReceiveLength := EOFIndex + EOFLength ; (*include count for EOF*)
				IF ((Index ) < InBufferDataLength) THEN
					MEMCPY(ADR(TempBuffer[0]),ADR(InBuffer[index]),DINT_TO_UDINT((InBufferDataLength-Index)));
					MEMSET( ADR(InBuffer),0,SIZEOF(InBuffer));
					InBufferDataLength := InBufferDataLength-Index;
					MEMCPY(ADR(InBuffer[0]),ADR(TempBuffer[0]),DINT_TO_UDINT(InBufferDataLength));
				ELSE
					MEMSET( ADR(InBuffer),0,SIZEOF(InBuffer));
					InBufferDataLength := 0;
				END_IF
				bDataAvailable := TRUE;
				EOFIndex := 0;
			END_IF
			State := 200;

		cFixedLength:		(*fixed receive lengh*)

			IF NOT bDataAvailable AND (InBufferDataLength >= MessageLength) THEN
				MEMCPY(pReceiveBuffer, ADR(InBuffer[0]),DINT_TO_UDINT(MessageLength)); (*copy data to output *)
				nReceiveLength := MessageLength;
				InBufferDataLength := InBufferDataLength - MessageLength;
				IF InBufferDataLength > 0 THEN
					(*still have data*)
					MEMCPY(ADR(TempBuffer[0]),ADR(InBuffer[MessageLength]),DINT_TO_UDINT(InBufferDataLength));
					MEMSET( ADR(InBuffer),0,SIZEOF(InBuffer));
					MEMCPY(ADR(InBuffer[0]),ADR(TempBuffer[0]),DINT_TO_UDINT(InBufferDataLength));
				ELSE
					MEMSET( ADR(InBuffer),0,SIZEOF(InBuffer));
					InBufferDataLength := 0;
				END_IF
				bDataAvailable := TRUE;
			END_IF
			State := 200;

		cContinuous:		(*continuous read*)
			State := 200;
		ELSE
			(*Software error*)
			bError := 1;
			sErrorText := 'Software error';
			State := 500;
	END_CASE;


300:	(*Copy Received Data Buffer*)
	IF  FirstEntry THEN
		bDataAvailable := FALSE;
		MEMSET(pReceiveBuffer,0,SIZEOF(pReceiveBuffer^));
		nReceiveLength := 0;
	END_IF

	IF NOT bReceived THEN
		IF InBufferDataLength > 0 THEN
			(*search again for another message*)
			State:=240;
		ELSE
			State:=200;
		END_IF
	END_IF

400:	(*Send Data If Any*)
	IF FirstEntry THEN
		fbSocketSend(bExecute:=FALSE);
		fbSocketSend(
			sSrvNetId := GVL.cNullString ,
			hSocket := hSocketHandle ,
			cbLen := DINT_TO_UDINT(TransmitLength+ 1),
			pSrc := pTransmitBuffer,
			bExecute := TRUE ,
			tTimeout := T#5s );
	END_IF
	IF NOT FirstEntry  THEN
		IF fbSocketSend.bBusy THEN
			bTransmitComplete := TRUE;
			State := 410;
		ELSIF fbSocketSend.bError THEN
			bError := 1;
			sErrorText := 'TCP/IP Send error';
			State := 500;
		END_IF
	END_IF

410:	(*Wait For Send Request To Go Low*)
	fbSocketSend(bExecute:=FALSE);
	IF NOT bSend THEN
		MEMSET(pTransmitBuffer,0,SIZEOF(pTransmitBuffer^));
		bTransmitComplete := FALSE;
		State := 200;
	END_IF

500:	(*Close Connection*)
	IF FirstEntry THEN
		fbSocketClose(bExecute:= FALSE);
		fbSocketClose(
			sSrvNetId := GVL.cNullString ,
			hSocket := hSocketHandle ,
			bExecute := TRUE,
			tTimeout := T#15s );
	END_IF
	tState500Timer(IN:=TRUE,PT:=T#1s);
	IF fbSocketClose.bBusy THEN
		tState500Timer(In:=FALSE);
		State := 510;
	END_IF
	IF tState500Timer.Q THEN
		tState500Timer(In:=FALSE);
		bError := TRUE;
		sErrorText := 'Socket Close Error: ';
		sErrorText := CONCAT(sErrorText, sRemoteHost);
		sErrorText := CONCAT(sErrorText,  ' Port ');
		sErrorText := CONCAT(sErrorText,  UDINT_TO_STRING(nRemotePort));
		State := 510;
	END_IF

510: (*Wait For Close*)
	fbSocketClose(bExecute:= FALSE);
	IF NOT fbSocketClose.bBusy THEN
		State := 0;
	END_IF

600: 	(*clear data*)

	IF  FirstEntry THEN
		MEMSET( ADR(InBuffer),0,SIZEOF(InBuffer));
		MEMSET(pTransmitBuffer,0,SIZEOF(pTransmitBuffer^));
		MEMSET(pReceiveBuffer,0,SIZEOF(pReceiveBuffer^));
		InBufferDataLength:=0;
		nErrorID:=0;
		bError:=FALSE;
		bDataAvailable:=FALSE;
		bTransmitComplete:=FALSE;
		bFlushComplete:=TRUE;
	END_IF
	IF NOT bFlush THEN
		bFlushComplete:=FALSE;
		State:=200;
	END_IF

END_CASE

(******END of sequence logic******)

END_FUNCTION_BLOCK

// POUs/Utility/F_GetTimeStamp
FUNCTION F_GetTimeStamp : TimeStamp
VAR_INPUT
END_VAR
VAR_OUTPUT
	gCurrentTime :TimeStamp;
END_VAR
VAR
	fbGetTime: GETSYSTEMTIME;
	TimeStamp:T_FileTime;
	CurrentTime: TIMESTRUCT;
	Time64 : T_ULarge_Integer;
	TimeShift : LREAL;
	TimeZoneOffset: DINT;
END_VAR

fbGetTime(timeLoDW=>Time64.dwLowPart , timeHiDW=>Time64.dwHighPart);
(*Correct for UTC time*)
(*Eastern Time zone*)
TimeZoneOffset := ABS(GVL.gTimeZoneOffsetFromUTC);
TimeShift := DINT_TO_LREAL(TimeZoneOffset) (*hours*) * DINT_TO_LREAL(3600) (*seconds*) * DINT_TO_LREAL(10000000) (*100ns*);
IF GVL.gTimeZoneOffsetFromUTC < 0 THEN
	Time64 := UInt64Sub64(Time64, LREAL_TO_UINT64(TimeShift));
ELSE
	Time64 := UInt64Add64(Time64, LREAL_TO_UINT64(TimeShift));
END_IF

TimeStamp.dwLowDateTime := Time64.dwLowPart;
TimeStamp.dwHighDateTime := Time64.dwHighPart;
CurrentTime := FILETIME_TO_SYSTEMTIME( TimeStamp );
F_GetTimeStamp.CurrentValue.dwHighPart := TimeStamp.dwHighDateTime;
F_GetTimeStamp.CurrentValue.dwLowPart := TimeStamp.dwLowDateTime;
F_GetTimeStamp.DateTime := CurrentTime;

END_FUNCTION

// POUs/Utility/FB_FileReadSettings
FUNCTION_BLOCK FB_FileReadSettings
VAR_INPUT
	pReadData	: POINTER TO BYTE;
	SizeOfData	: UDINT;
	FileName	: T_MaxString;  	(* file path and name *)
	bExecute	: BOOL;		(* rising edge starts fb execution *)
END_VAR
VAR_OUTPUT
	bError		:BOOL;
	bDone		:BOOL;
END_VAR
VAR
	nErrId		:UDINT;
	bBusy		:BOOL;
	fbFileOpen	:FB_FileOpen;
	fbFileClose	:FB_FileClose;
	fbFileRead	:FB_FileRead;

	hFile		:UINT	:= 0;(* file handle of the file *)

	Step		:DWORD;
	RisingEdge	:R_TRIG;

	cbReadLength	:UDINT:=0;
END_VAR

RisingEdge(CLK:=bExecute);
IF RisingEdge.Q THEN
	IF NOT bBusy THEN
		bBusy := TRUE;
		bError:= FALSE;
		nErrId:=0;
		Step := 1;
		cbReadLength:=0;
		hFile:=0;
		MEMSET(pReadData, 0, SizeOfData); (* Clear the data before we really read it *)
	END_IF
END_IF

bDone := NOT bBusy AND bExecute;
bError := bError AND bExecute;

CASE Step OF
	0:(* do nothing *)
	;

	1:(* open file *)
	fbFileOpen(  bExecute := FALSE  );
	fbFileOpen(	sNetId := '',
		sPathName := FileName,
		nMode := FOPEN_MODEREAD OR FOPEN_MODEBINARY,
		ePath := PATH_GENERIC,
		tTimeout := T#2s,
		bExecute := TRUE );
		Step := Step + 1;

	2:
	fbFileOpen( bExecute := FALSE );
	IF ( NOT fbFileOpen.bBusy ) THEN
		IF ( fbFileOpen.bError ) THEN
			nErrId := fbFileOpen.nErrId;
			bError := TRUE;
			Step := 50;
		ELSE
			hFile := fbFileOpen.hFile;
			Step := 5;
		END_IF
	END_IF

	5:(*read data from source file*)
	cbReadLength := 0;
	fbFileRead( bExecute:= FALSE );
	fbFileRead( 	sNetId:='',
			hFile:=hFile,
			pReadBuff:= pReadData,
			cbReadLen:= SizeOfData,
			bExecute:=TRUE,
			tTimeout:=T#2s );
	Step := Step + 1;

	6:
	fbFileRead( bExecute:= FALSE );
	IF ( NOT fbFileRead.bBusy ) THEN
		IF ( fbFileRead.bError ) THEN
			nErrId := fbFileRead.nErrId;
			bError := TRUE;
			Step := 50;
		ELSIF fbFileRead.cbRead <> SizeOfData THEN
			nErrId := fbFileRead.nErrId;
			bError := TRUE;
			Step := 50;
		ELSE
			cbReadLength := fbFileRead.cbRead;
			Step := 50;
		END_IF
	END_IF


	30:(* close the file *)
	fbFileClose( bExecute := FALSE );
	fbFileClose( 	sNetId:='',
			hFile:=hFile,
			bExecute:=TRUE,
			tTimeout:=T#2s );
	Step := Step + 1;

	31:
	fbFileClose( bExecute := FALSE );
	IF ( NOT fbFileClose.bBusy ) THEN
		IF ( fbFileClose.bError ) THEN
			nErrId := fbFileClose.nErrId;
			bError := TRUE;
		END_IF
		Step := 50;
		hFile := 0;
	END_IF


	50: (*error or ready => cleanup*)
	IF ( hFile <> 0 ) THEN
		Step := 30; (* close the file*)
	ELSE
		Step := 0;	(* ready *)
		bBusy := FALSE;
	END_IF

END_CASE

END_FUNCTION_BLOCK

// POUs/Utility/FB_FileWriteSettings
FUNCTION_BLOCK FB_FileWriteSettings
VAR_INPUT
	pDataToWrite: POINTER TO BYTE;
	SizeOfData	: UDINT;
	FileName	: T_MaxString;  	(* file path and name *)
	bExecute	: BOOL;		(* rising edge starts fb execution *)
END_VAR
VAR_OUTPUT
	bError		:BOOL;
	bDone		:BOOL;
END_VAR
VAR
	nErrId		:UDINT;
	bBusy: BOOL;
	fbFileOpen	:FB_FileOpen;
	fbFileClose	:FB_FileClose;
	fbFileWrite	:FB_FileWrite;

	hFile		:UINT	:= 0;(* file handle of the  file *)

	Step		:DWORD;
	RisingEdge	:R_TRIG;
END_VAR

RisingEdge(CLK:=bExecute);
IF RisingEdge.Q THEN
	IF NOT bBusy THEN
		bBusy := TRUE;
		bError:= FALSE;
		nErrId:=0;
		Step := 3;
		hFile:=0;
	END_IF
END_IF

bDone := NOT bBusy AND bExecute;
bError := bError AND bExecute;

CASE Step OF
	0:(* do nothing *)
	;

	3:(* open  file *)
	fbFileOpen(  bExecute := FALSE  );
	fbFileOpen( 	sNetId := '',
			sPathName := FileName,
			nMode := FOPEN_MODEWRITE OR FOPEN_MODEBINARY,
			ePath := PATH_GENERIC,
			tTimeout := T#2s,
			bExecute := TRUE );
	Step := Step+1;

	4:
	fbFileOpen(  bExecute := FALSE  );
	IF ( NOT fbFileOpen.bBusy ) THEN
		IF ( fbFileOpen.bError ) THEN
			nErrId := fbFileOpen.nErrId;
			bError := TRUE;
			Step := 50;
		ELSE
			hFile := fbFileOpen.hFile;
			Step := 7;
		END_IF
	END_IF

	7:(*write data to  file*)
	fbFileWrite( bExecute := FALSE );
	fbFileWrite(	sNetId:='',
			hFile:=hFile,
			pWriteBuff:= pDataToWrite,
			cbWriteLen:= SizeOfData,
			bExecute:=TRUE,
			tTimeout:=T#2s );
	Step := Step + 1;

	8:
	fbFileWrite( bExecute := FALSE );
	IF ( NOT fbFileWrite.bBusy ) THEN
		IF ( fbFileWrite.bError ) THEN
			nErrId := fbFileWrite.nErrId;
			bError := TRUE;
			Step := 50;
		ELSE
			Step := 50;(*cleanup: close the file *)
		END_IF
	END_IF

	30:(* close the file *)
	fbFileClose( bExecute := FALSE );
	fbFileClose( 	sNetId:='',
			hFile:=hFile,
			bExecute:=TRUE,
			tTimeout:=T#2s );
	Step := Step + 1;

	31:
	fbFileClose( bExecute := FALSE );
	IF ( NOT fbFileClose.bBusy ) THEN
		IF ( fbFileClose.bError ) THEN
			nErrId := fbFileClose.nErrId;
			bError := TRUE;
		END_IF
		Step := 50;
		hFile := 0;
	END_IF


	50: (*error or ready => cleanup*)
	IF ( hFile <> 0 ) THEN
		Step := 30; (* close the destination file*)
	ELSE
		Step := 0;	(* ready *)
		bBusy := FALSE;
	END_IF

END_CASE

END_FUNCTION_BLOCK

// POUs/Utility/FB_Sensor
FUNCTION_BLOCK FB_Sensor
VAR_INPUT
    Reset : BOOL := TRUE;
    Input : BOOL := FALSE;

    OnTime : TIME := T#0.0S;
    OffTime : TIME := T#0.0S;
END_VAR
VAR_OUTPUT
    On : BOOL := FALSE;
    Off : BOOL := FALSE;
END_VAR
VAR
    tmrOn : TON;
    tmrOff : TON;
END_VAR

(*  reset the timer (i.e. IN := FALSE) anytime bReset is TRUE;*)

     IF Reset OR Gvl.gFirstScan THEN
        tmrOn(IN := FALSE);
        tmrOff(IN := FALSE);
        On := FALSE;
        Off := FALSE;
        Reset := FALSE;
        RETURN;
    END_IF;

    tmrOn(IN := Input, PT := OnTime);
    On := tmrOn.Q;

    tmrOff(IN := (NOT Input), PT := OffTime);
    Off := tmrOff.Q;

END_FUNCTION_BLOCK

// POUs/Utility/FIFO_DINT100
FUNCTION_BLOCK FIFO_DINT100
VAR_INPUT
	Overwrite	: BOOL;
	pFIFO		: POINTER TO Dint100FIFOBuffer;
	in			: DINT;
END_VAR
VAR_OUTPUT
	Err		: BOOL;
	Count	: DINT;
	Full		: BOOL;
	out		: DINT;
END_VAR
VAR
	Head : DINT;
	Tail: DINT;
	Idx: DINT;
END_VAR

ACTION INIT:
idx := pFIFO^.Size * SIZEOF(in);
MEMSET(ADR( pFIFO^.Buffer[0]), 0, DINT_TO_UDINT(idx));
MEMSET(ADR(in),0,SIZEOF(in));
MEMSET(ADR(out),0,SIZEOF(out));
Count:=0;
Head:=0;
Tail:=0;
Full:=0;
Err:=0;
END_ACTION

ACTION INSERT:
Err := 0;
IF (Full AND Overwrite) OR NOT Full THEN
	pFIFO^.buffer[Head]:=in;
	Head := Head + 1;
	IF Head = pFIFO^.Size THEN
		Head:=0;
	END_IF
	IF Full THEN
		Tail := Tail +1;
		IF Tail = pFIFO^.Size THEN
			Tail :=0;
		END_IF
	ELSE
		Count := Count  +1;
	END_IF
ELSE
	err:=1;
END_IF
Full := (Head = Tail);
END_ACTION

ACTION PEEK:
err:=0;
IF Full OR (Tail <> Head) THEN
	out := pFIFO^.buffer[Tail];
ELSE
	err:=1; (*fifo is empty*)
END_IF
END_ACTION

ACTION REMOVE:
err:=0;
IF NOT Full AND (Head = Tail) THEN
	(*empty*)
	err:=1;
ELSE
	out := pFIFO^.Buffer[Tail];
	MEMSET(ADR(pFIFO^.buffer[Tail]), 0, SIZEOF (in));
	Tail := Tail +1;
	Count := Count  - 1;
	IF Tail = pFIFO^.Size THEN
		Tail := 0;
	END_IF
	Full := 0;
END_IF
END_ACTION

END_FUNCTION_BLOCK

// POUs/Utility/FIFO_ID50
FUNCTION_BLOCK FIFO_ID50
VAR_INPUT
	Overwrite	: BOOL;
	pFIFO		: POINTER TO ID50FIFOBuffer;
	in			: ComponentIdentifier;
END_VAR
VAR_OUTPUT
	Err		: BOOL;
	Count	: DINT;
	Full		: BOOL;
	out		: ComponentIdentifier;
END_VAR
VAR
	Head : DINT;
	Tail: DINT;
	Idx: DINT;
END_VAR

ACTION INIT:
idx := pFIFO^.Size * SIZEOF(in);
MEMSET(ADR( pFIFO^.Buffer[0]), 0, DINT_TO_UDINT(idx));
MEMSET(ADR(in),0,SIZEOF(in));
MEMSET(ADR(out),0,SIZEOF(out));
Count:=0;
Head:=0;
Tail:=0;
Full:=0;
Err:=0;
END_ACTION

ACTION INSERT:
Err := 0;
IF (Full AND Overwrite) OR NOT Full THEN
	pFIFO^.buffer[Head]:=in;
	Head := Head + 1;
	IF Head = pFIFO^.Size THEN
		Head:=0;
	END_IF
	IF Full THEN
		Tail := Tail +1;
		IF Tail = pFIFO^.Size THEN
			Tail :=0;
		END_IF
	ELSE
		Count := Count  +1;
	END_IF
ELSE
	err:=1;
END_IF
Full := (Head = Tail);
END_ACTION

ACTION PEEK:
err:=0;
IF Full OR (Tail <> Head) THEN
	out := pFIFO^.buffer[Tail];
ELSE
	err:=1; (*fifo is empty*)
END_IF
END_ACTION

ACTION REMOVE:
err:=0;
IF NOT Full AND (Head = Tail) THEN
	(*empty*)
	err:=1;
ELSE
	out := pFIFO^.Buffer[Tail];
	MEMSET(ADR(pFIFO^.buffer[Tail]), 0, SIZEOF (in));
	Tail := Tail +1;
	Count := Count  - 1;
	IF Tail = pFIFO^.Size THEN
		Tail := 0;
	END_IF
	Full := 0;
END_IF
END_ACTION

END_FUNCTION_BLOCK

// POUs/Utility/FIFO_LREAL100
FUNCTION_BLOCK FIFO_LREAL100
VAR_INPUT
	Overwrite	: BOOL;
	pFIFO		: POINTER TO LREAL100FIFOBuffer;
	in			: LREAL;
END_VAR
VAR_OUTPUT
	Err		: BOOL;
	Count	: DINT;
	Full		: BOOL;
	out		: LREAL;
END_VAR
VAR
	Head : DINT;
	Tail: DINT;
	Idx: DINT;
END_VAR

ACTION INIT:
idx := pFIFO^.Size * SIZEOF(in);
MEMSET(ADR( pFIFO^.Buffer[0]), 0, DINT_TO_UDINT(idx));
MEMSET(ADR(in),0,SIZEOF(in));
MEMSET(ADR(out),0,SIZEOF(out));
Count:=0;
Head:=0;
Tail:=0;
Full:=0;
Err:=0;
END_ACTION

ACTION INSERT:
Err := 0;
IF (Full AND Overwrite) OR NOT Full THEN
	pFIFO^.buffer[Head]:=in;
	Head := Head + 1;
	IF Head = pFIFO^.Size THEN
		Head:=0;
	END_IF
	IF Full THEN
		Tail := Tail +1;
		IF Tail = pFIFO^.Size THEN
			Tail :=0;
		END_IF
	ELSE
		Count := Count  +1;
	END_IF
ELSE
	err:=1;
END_IF
Full := (Head = Tail);
END_ACTION

ACTION PEEK:
err:=0;
IF Full OR (Tail <> Head) THEN
	out := pFIFO^.buffer[Tail];
ELSE
	err:=1; (*fifo is empty*)
END_IF
END_ACTION

ACTION REMOVE:
err:=0;
IF NOT Full AND (Head = Tail) THEN
	(*empty*)
	err:=1;
ELSE
	out := pFIFO^.Buffer[Tail];
	MEMSET(ADR(pFIFO^.buffer[Tail]), 0, SIZEOF (in));
	Tail := Tail +1;
	Count := Count  - 1;
	IF Tail = pFIFO^.Size THEN
		Tail := 0;
	END_IF
	Full := 0;
END_IF
END_ACTION

END_FUNCTION_BLOCK

// POUs/Utility/LEFTBigString
FUNCTION LEFTBigString : BOOL

	VAR_INPUT
	pInputString		: POINTER TO BYTE;
	SizeOfInputString	: UINT;
	SizeToCopy			: UINT;
	pOutputString		: POINTER TO BYTE;
	SizeOfOutputString	: UINT;
END_VAR
VAR
	i					: INT;
	pOutputStringNull	: POINTER TO BYTE;
END_VAR

(* Make sure output string is big enough to hold the characters *)
IF SizeOfOutputString < SizeToCopy THEN
	RETURN;
END_IF

(* Copy bytes from input string to output string *)
MEMCPY(pOutputString, pInputString, SizeToCopy);

(* Append null character to end of output string *)
pOutputStringNull := (pOutputString + SizeToCopy);
pOutputStringNull^ := 0;
LEFTBigString:= TRUE;

END_FUNCTION

// POUs/Utility/RIGHTBigString
FUNCTION RIGHTBigString : BOOL
VAR_INPUT
	pInputString					: POINTER TO BYTE;
	SizeOfInputString				: UINT;
	SizeToCopy						: UINT;
	pOutputString					: POINTER TO BYTE;
	SizeOfOutputString				: DINT;
END_VAR
VAR
	i								: DINT;
	pInputStringNull				: POINTER TO BYTE;
	pOutputStringNull				: POINTER TO BYTE;
	NumberOfInputStringCharacters	: DINT;
END_VAR

(* Make sure output string is big enough to hold the characters *)
IF SizeOfOutputString < SizeToCopy THEN
	RETURN;
END_IF

(* Find address of null character for input string *)
pInputStringNull := pInputString;
FOR i := 0 TO SizeOfInputString DO
	IF pInputStringNull^ = 0 THEN
		EXIT;
	END_IF
	pInputStringNull := pInputStringNull + 1;
END_FOR

(* Check to see if there are enough characters in input string, otherwise copy them all *)
NumberOfInputStringCharacters := (SIZEOF(pInputStringNull) - SIZEOF(pInputString));
IF NumberOfInputStringCharacters < UINT_TO_DINT(SizeToCopy) THEN
	(* Copy bytes from input string to output string *)
	MEMCPY(pOutputString, (SIZEOF(pInputStringNull) - NumberOfInputStringCharacters), DINT_TO_UDINT(NumberOfInputStringCharacters));

	(* Append null character to end of output string *)
	pOutputStringNull := (pOutputString + SIZEOF(NumberOfInputStringCharacters));
	pOutputStringNull^ := 0;
	RETURN;
END_IF

(* Copy bytes from input string to output string *)
MEMCPY(pOutputString, SIZEOF(pInputStringNull) - UINT_TO_DINT(SizeToCopy), SizeToCopy);

(* Append null character to end of output string *)
pOutputStringNull := (pOutputString + UINT_TO_DINT(SizeToCopy));
pOutputStringNull^ := 0;

RIGHTBigString:=TRUE;

END_FUNCTION

// POUs/MAIN
PROGRAM MAIN
VAR
END_VAR

END_PROGRAM
